(* IEC 61131-3 sources: inproshop/Team-Test20_exported/OP80/2.PRG, 7 files *)

(* ---- OP80_Communication.st ---- *)
PROGRAM OP80_Communication
VAR
	HeartdelayON:TON;
	HeartdelayOFF:TON;
	MasterHeartdelayON:TON;
	MasterHeartdelayOFF:TON;
END_VAR

//心跳输出
IF CPU_Clock.Clock_1s THEN
	DB8005_Communication.TO_OPXX.Heart:=1;
ELSE
	DB8005_Communication.TO_OPXX.Heart:=0;
END_IF
//给前站安全信号
IF NOT DB8050_DriveControl.KUKA[1].Status.InterFace_B[49]  OR DB8000_Control.Mode.Status.OfflineMode THEN
	DB8005_Communication.TO_OPXX.Safe:=1;
ELSE
	DB8005_Communication.TO_OPXX.Safe:=0;
END_IF;

HeartdelayON(IN:= DB8005_Communication.TO_OPXX.Heart=1, PT:= T#2S, Q=> , ET=> );
HeartdelayOFF(IN:= DB8005_Communication.TO_OPXX.Heart=0, PT:= T#2S, Q=> , ET=> );
//前站掉线报警
IF (HeartdelayON.Q OR HeartdelayOFF.Q) AND NOT DB8000_Control.Mode.Status.OfflineMode  THEN
	DB8070_Fault.Stop.BeforStation_Communication_Rrror:=TRUE;
END_IF

//主站心跳通讯检测
MasterHeartdelayON(IN:= DB8005_Communication.FromMaster.Heart=1, PT:= T#2S, Q=> , ET=> );
MasterHeartdelayOFF(IN:= DB8005_Communication.FromMaster.Heart=0, PT:= T#2S, Q=> , ET=> );
//主站掉线报警
IF (MasterHeartdelayON.Q OR MasterHeartdelayOFF.Q) AND NOT DB8000_Control.Mode.Status.OfflineMode  THEN
	DB8070_Fault.Stop.MasterTimeOut:=TRUE;
END_IF

//与主站配方不一致报警
IF DB8005_Communication.FromMaster.MasterRecipeID<>DB8002_Recipe.RecipeNum AND NOT DB8000_Control.Mode.Status.OfflineMode THEN
	DB8070_Fault.Stop.MaterReipeDiscrepancy:=TRUE;
END_IF

(* ---- OP80_DI_Mirror.st ---- *)
PROGRAM OP80_DI_Mirror
VAR
	i:INT;//循环用变量
	Page:INT;
	Monitor:ARRAY[0..15] OF Str_IOMonitor;
	Status:WORD;
	Map:BOOL;
END_VAR

ACT_MAP();
ACT_Comment();
ACT_Status();

(* ---- OP80_DO_Mirror.st ---- *)
PROGRAM OP80_DO_Mirror
VAR
	i:INT;//循环用变量
	Page:INT;
	Monitor:ARRAY[0..15] OF Str_IOMonitor;
	Status:WORD;
	Map:BOOL;
	Startlamp1:BOOL;
	Startlamp2:BOOL;
END_VAR

ACT_MAP();
ACT_Comment();
ACT_Status();

(* ---- OP80_DriveControl.st ---- *)
PROGRAM OP80_DriveControl
VAR
	FB_Cylinder_instance :ARRAY[0..63]OF FB_Cylinder_V1;
	FB_Vacuum_instance :ARRAY[0..31]OF FB_Vacuum_V1;
	FB_Axis_Instance:ARRAY[0..31]OF FB_Axis_V1_3;
	FB_Sensor_instance :ARRAY[0..200]OF FB_Sensor_V1_1;
	FB_TcpClient_Instance:ARRAY[0..31]OF FB_TcpClient;
	FB_DoubleStart_Instance:ARRAY[1..4]OF FB_DoubleStart;
	FB_Epson_V1_Instance:ARRAY[1..1]OF FB_Epson_V1;
	FB_Kuka_V1_Instance:ARRAY[1..2]OF FB_Kuka6_V1;
	FB_Rotdisk_V1_Instance:ARRAY[1..1]OF FB_Rotdisk_V1;
	FB_Stopper_V1_Instance:ARRAY[1..1]OF FB_Stopper_V1;
	FB_AI_Instance:ARRAY[1..200]OF FB_AI;
	FB_Motor_Instance:ARRAY[1..1]OF FB_Motor;
	FB_Heating_Instance:ARRAY[1..1]OF FB_Heating;
	FB_Gear_Instance:ARRAY[1..1]OF FB_Gear;
	FB_AAS_Instance:ARRAY[1..1]OF FB_AAS;
	FB_Aging_Instance:ARRAY[1..80]OF FB_Aging;
	FB_AirLeak_Instance:ARRAY[1..2]OF FB_AirLeak;
	FB_Palletizing_Instance:ARRAY[1..3]OF FB_Palletizing;
END_VAR
VAR
	i:INT;//循环变量用
	j:INT;//循环变量用
END_VAR

VAR
	TempKUKA1InPut AT %IB4500:ARRAY[0..63]OF BYTE;
	TempKUKA1OutPut AT %QB4500:ARRAY[0..63]OF BYTE;
	TempKUKA2InPut AT %IB4600:ARRAY[0..63]OF BYTE;
	TempKUKA2OutPut AT %QB4600:ARRAY[0..63]OF BYTE;
END_VAR
VAR
	PowerLimitDelay:ARRAY[0..16] OF TON;//超出额定电流
END_VAR

ACT_Axis();
ACT_Cylinder();
ACT_Vacuum();
ACT_Epson();
ACT_Kuka();
ACT_Sensor();
ACT_Motor();
ACT_Rotdisk();
ACT_AI();
ACT_Stopper();

ACT_Pallet();

(* ---- OP80_Fault.st ---- *)
PROGRAM OP80_Fault
VAR
	i:UINT;//循环变量用
	Pobool_IN: POINTER TO BOOL;//输入报警指针地址获取；
	Pobool_OUT: POINTER TO BOOL;//输出报警指针地址获取；
	EstopMAP:ARRAY[0..255] OF BOOL;
	StopMAP:ARRAY[0..999] OF BOOL;
	RunMAP:ARRAY[0..255] OF BOOL;
	Size:UINT;//数组数量
	Estop_R:R_TRIG;//急停上升沿
	Stop_R:R_TRIG;//暂停上升沿
	Run_R:R_TRIG;//警告上升沿
	StopFaultDelay:ARRAY[1..10]OF TON;//停止报警延时
END_VAR

//气缸报警地址映射
SizeOfAry(In:=DB8050_DriveControl.CylCtrl,Out=>Size);
FOR i:=0 TO Size-1 BY 1 DO
	DB8070_Fault.Stop.Cyl[I]:=DB8050_DriveControl.CylCtrl[i].Status.Error;
END_FOR
//真空报警映射
SizeOfAry(In:=DB8050_DriveControl.VacCtrl,Out=>Size);
FOR i:=0 TO Size-1 BY 1 DO
	DB8070_Fault.Stop.Vac[I]:=DB8050_DriveControl.VacCtrl[i].Status.Error;
END_FOR
//轴报警映射
SizeOfAry(In:=DB8050_DriveControl.AxisCtrl,Out=>Size);
FOR i:=0 TO Size-1 BY 1 DO
	DB8070_Fault.Stop.Axis[I]:=DB8050_DriveControl.AxisCtrl[i].Status.Error;
END_FOR

//急停报警
DB8070_Fault.Estop.EstopButton:=NOT DB8000_Control.Machine.EmgSafetyRelay;

//暂停故障

//提示

ACT_MAP();
ACT_HMI_Jump();

(* ---- OP80_Graph.st ---- *)
PROGRAM OP80_Graph
VAR
	IntitalTimeDelay:ARRAY[1..9,0..10] OF TON;//初始化流程用
	AutoTimeDelay:ARRAY[1..9,0..10] OF TON;//自动流程用

	Init:ARRAY[1..20]OF Str_Graph := [20((Complete := TRUE))];//初始化
	Auto:ARRAY[1..20]OF Str_Graph;//自动
	Start:ARRAY[1..9] OF BOOL;//自动启动条件
	i:INT;//循环变量用

END_VAR

ACT_InitST1();
ACT_InitST2();
ACT_InitST3();
ACT_InitST4();

ACT_AutoRunST1_气密1测试();
ACT_AutoRunST2_气密2测试();
ACT_AutoRunST3_气密3测试();
ACT_AutoRunST4_气密4测试();

(* ---- OP80_Other.st ---- *)
PROGRAM OP80_Other
VAR
	i:INT;//循环变量
	MaterialCode: INT;
END_VAR

//产品1
DB8090_Other.Product[1].ProductSpecifications:='  ';
DB8090_Other.Product[1].ProductCode:=' ';

DB8090_Other.Product[1].MaterialCode[1]:=' ';
DB8090_Other.Product[1].MaterialCode[2]:=' ';

//产品2
DB8090_Other.Product[2].ProductSpecifications:=' ';
DB8090_Other.Product[2].ProductCode:=' ';

DB8090_Other.Product[2].MaterialCode[1]:=' ';
DB8090_Other.Product[2].MaterialCode[2]:=' ';

//产品3_S20LW-2
DB8090_Other.Product[3].ProductSpecifications:=' ';
DB8090_Other.Product[3].ProductCode:=' ';

DB8090_Other.Product[3].MaterialCode[1]:=' ';
DB8090_Other.Product[3].MaterialCode[2]:=' ';

FOR i:=1 TO 20 BY 1 DO
	DB8090_Other.Product[i].MaterialName[1]:=" ";
	DB8090_Other.Product[i].MaterialName[2]:=" ";
END_FOR

//产品对应编号检索
FOR i:=1 TO 20 BY 1 DO
	IF DB8002_Recipe.TypeData[DB8002_Recipe.RecipeNum].Name=DB8090_Other.Product[i].ProductSpecifications THEN
		DB8002_Recipe.TypeData[DB8002_Recipe.RecipeNum].ProDuctNum:=i;
		EXIT;
	END_IF

END_FOR
IF i>=21 THEN
	;
END_IF

//动作分类
IF DB8090_Other.Product[DB8002_Recipe.TypeDataCur.ProDuctNum].MaterialCode[1]='PGH64' THEN
	DB8090_Other.Cyl_B_Sport:=TRUE;
ELSE
	DB8090_Other.Cyl_B_Sport:=FALSE;
END_IF
